// TIA Portal V16 export
// export: Created 2022-03-06T01:16:19.959555Z, ExportSetting WithDefaults, DisplayName Totally Integrated Automation Portal, DisplayVersion V16 Update 4, DisplayName TIA Portal Version Control Interface, DisplayVersion V16 Update 2, DisplayName TIA Portal Openness, DisplayVersion V16 Update 4, DisplayName TIA Portal Teamcenter Gateway, DisplayVersion V16, DisplayName SINAMICS Startdrive Advanced, DisplayVersion V16 Update 4, DisplayName SINAMICS Startdrive G110M, G120, G120C, G120D, G120P, G115D, DisplayVersion V16 Update 4, DisplayName SINAMICS Startdrive G130, G150, S120, S150, SINAMICS MV, S210, DisplayVersion V16 Update 4, DisplayName STEP 7 Professional, DisplayVersion V16 Update 4, DisplayName STEP 7 Safety, DisplayVersion V16, DisplayName WinCC Advanced / Unified PC, DisplayVersion V16 Update 4
FUNCTION "Escalamiento" : Void   // FC1, LAD
{ S7_Optimized_Access := 'TRUE' }
VERSION : 0.1
// stored: AutoNumber true, IsIECCheckEnabled false, SetENOAutomatically false, UDAEnableTagReadback false
   VAR_INPUT
      EntradaTx : Int;
      Minimo : Real;
      Maximo : Real;
   END_VAR
   VAR_OUTPUT
      SalidaEscalada : Real;
   END_VAR
   VAR_TEMP
      entrada_norm : Real;
   END_VAR
BEGIN

REGION Network 1
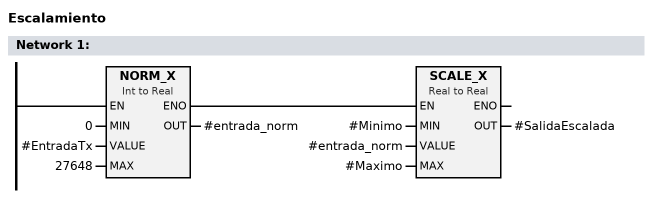
   RUNG wire#powerrail
      { S7_Templates := "[SrcType := Int, DestType := Real]" } Normalize(min := 0, value := #EntradaTx, max := 27648, out => #entrada_norm)
      { S7_Templates := "[SrcType := Real, DestType := Real]" } Scale(min := #Minimo, value := #entrada_norm, max := #Maximo, out => #SalidaEscalada)
   END_RUNG
   // the same network as SCL:
   #entrada_norm := NORM_X(MIN := 0, VALUE := #EntradaTx, MAX := 27648);
   #SalidaEscalada := SCALE_X(MIN := #Minimo, VALUE := #entrada_norm, MAX := #Maximo);
END_REGION
END_FUNCTION
